FUNCTION_BLOCK Test_TEvent_AddEventHandler_IncsNumberOfEventHandlers EXTENDS TUnitTestbase
VAR
    TestEvent : TTestEvent;
    TestEventHandler : TTestEventHandler;
END_VAR



TestEvent
    .ClearEventHandlers()
    .AddEventHandler(TestEventHandler);
    
Assertion.AssertEquals_UDINT(
    Expected := 1,
    Actual   := TestEvent.EventHandlers.Count,
    VariableName  := 'TestEvent.EventHandlers.Count');
    

TestFinished();

END_FUNCTION_BLOCK

(* stored: Version 1.1.0.1, ProductVersion 3.1.4024.4
   POU Test_TEvent_AddEventHandler_IncsNumberOfEventHandlers: Id {3a9e060b-7494-4c68-a9ca-d469d88b76ad}, SpecialFunc None *)
